FUNCTION_BLOCK L3_ProcessPlan (* Composite Function Block Type *)
  (* Standard: 61499-2 *)
  (* Version 0.0, 2014-10-13, EQUEROL, UJI *)
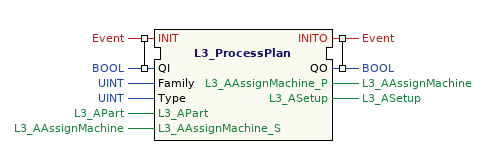
  EVENT_INPUT
    INIT WITH QI; (* Initialization Request *)
  END_EVENT
  EVENT_OUTPUT
    INITO WITH QO; (* Initialization Confirm *)
  END_EVENT
  VAR_INPUT
    QI : BOOL; (* Input event qualifier *)
    Family : UINT; (* Process plan family *)
    Type : UINT; (* Process plan type *)
  END_VAR
  VAR_OUTPUT
    QO : BOOL; (* Output event qualifier *)
  END_VAR
  SOCKETS
    L3_APart : L3_APart;
    L3_AAssignMachine_S : L3_AAssignMachine;
  END_SOCKETS
  PLUGS
    L3_AAssignMachine_P : L3_AAssignMachine;
    L3_ASetup : L3_ASetup;
  END_PLUGS
  FBS
    L3_PPTable : L3_PPTable;
    L3_NewPartHDLR : L3_NewPartHDLR;
    L3_MachineAllocator : L3_MachineAllocator;
    L3_MachineChecker : L3_MachineChecker;
    L3_CompletedPartHDLR : L3_CompletedPartHDLR;
    E_DELAY : E_DELAY;
    L3_SetupTable : L3_SetupTable;
    E_DELAY_1 : E_DELAY;
    L3_CompletedSetupHDLR_1 : L3_CompletedSetupHDLR;
  END_FBS
  EVENT_CONNECTIONS
    L3_AAssignMachine_S.CHK TO L3_MachineChecker.REQ;
    L3_MachineChecker.IND TO L3_PPTable.REQ;
    L3_PPTable.CNF TO L3_MachineChecker.RSP;
    L3_MachineChecker.CNF TO L3_AAssignMachine_P.CHK;
    L3_AAssignMachine_S.ASG TO L3_MachineAllocator.REQ;
    L3_MachineAllocator.Start TO E_DELAY.START;
    L3_MachineAllocator.Stop TO E_DELAY.STOP;
    E_DELAY.EO TO L3_MachineAllocator.Timeout;
    L3_MachineAllocator.CNF TO L3_AAssignMachine_P.ASG;
    L3_MachineAllocator.IND1 TO L3_SetupTable.REQ;
    L3_ASetup.CNF TO L3_MachineAllocator.RSP1;
    L3_MachineAllocator.IND2 TO L3_PPTable.REQ2;
    L3_PPTable.CNF2 TO L3_MachineAllocator.RSP2;
    L3_PPTable.CNF TO L3_MachineAllocator.REQ2;
    L3_SetupTable.CNF TO L3_ASetup.REQ;
    L3_APart.REQ TO L3_NewPartHDLR.REQ1;
    L3_NewPartHDLR.CNF1 TO L3_APart.CNF;
    L3_PPTable.IND1 TO L3_NewPartHDLR.REQ2;
    L3_NewPartHDLR.CNF2 TO L3_PPTable.RSP1;
    L3_CompletedPartHDLR.Start TO E_DELAY_1.START;
    L3_CompletedPartHDLR.Stop TO E_DELAY_1.STOP;
    E_DELAY_1.EO TO L3_CompletedPartHDLR.Timeout;
    L3_CompletedPartHDLR.CNF TO L3_PPTable.RSP3;
    L3_PPTable.IND3 TO L3_CompletedPartHDLR.REQ;
    L3_CompletedPartHDLR.IND TO L3_APart.IND;
    L3_APart.RSP TO L3_CompletedPartHDLR.RSP;
    L3_CompletedPartHDLR.INITO TO L3_PPTable.INIT;
    INIT TO L3_CompletedPartHDLR.INIT;
    L3_PPTable.INITO TO L3_SetupTable.INIT;
    L3_SetupTable.INITO TO INITO;
    L3_CompletedSetupHDLR_1.CNF1 TO L3_PPTable.RSP2;
    L3_PPTable.IND2 TO L3_CompletedSetupHDLR_1.REQ1;
    L3_ASetup.IND TO L3_CompletedSetupHDLR_1.REQ;
    L3_CompletedSetupHDLR_1.CNF TO L3_ASetup.RSP;
  END_CONNECTIONS
  DATA_CONNECTIONS
    L3_AAssignMachine_S.MTypeP TO L3_MachineChecker.MTypeIn;
    L3_AAssignMachine_S.MStateP TO L3_MachineChecker.MStateIn;
    L3_AAssignMachine_S.MPriorityP TO L3_MachineChecker.MPriorityIn;
    L3_AAssignMachine_S.MAssignP TO L3_MachineChecker.MAssignIn;
    L3_MachineChecker.MTypeOut TO L3_AAssignMachine_P.MTypeP;
    L3_MachineChecker.MStateOut TO L3_AAssignMachine_P.MStateP;
    L3_MachineChecker.MPriorityOut TO L3_AAssignMachine_P.MPriorityP;
    L3_MachineChecker.MAssignOut TO L3_AAssignMachine_P.MAssignP;
    L3_PPTable.vPriority TO L3_MachineChecker.Priority;
    L3_MachineAllocator.Delay TO E_DELAY.DT;
    L3_AAssignMachine_S.MFinalAssignP TO L3_MachineAllocator.MFinalAssignIn;
    L3_MachineAllocator.MFinalAssignOut TO L3_AAssignMachine_P.MFinalAssignP;
    L3_PPTable.vPartIDOut TO L3_MachineChecker.PartID;
    L3_PPTable.vPartIDOut TO L3_MachineAllocator.PartIDIn;
    L3_PPTable.vSetup TO L3_MachineAllocator.SetupIDIn;
    L3_MachineAllocator.PartIDOut TO L3_SetupTable.PartID;
    L3_MachineAllocator.SetupID TO L3_SetupTable.SetupID;
    L3_MachineAllocator.MID TO L3_SetupTable.MID;
    L3_SetupTable.PartInfo TO L3_ASetup.PartInfoP;
    L3_SetupTable.MID2 TO L3_ASetup.MID;
    L3_SetupTable.OPIDS TO L3_ASetup.OPIDS;
    L3_SetupTable.OPParams TO L3_ASetup.OPParams;
    L3_SetupTable.Fixture TO L3_ASetup.Fixture;
    L3_MachineAllocator.PartIDOut TO L3_PPTable.PartIDIn3;
    L3_MachineAllocator.MID TO L3_PPTable.MID;
    L3_APart.PartIDP TO L3_NewPartHDLR.PartIDIn;
    L3_APart.Lotsize TO L3_NewPartHDLR.LotsizeIn;
    L3_APart.Deadline TO L3_NewPartHDLR.DeadlineIn;
    L3_NewPartHDLR.PartIDOut TO L3_PPTable.PartIDIn1;
    L3_NewPartHDLR.LotsizeOut TO L3_PPTable.LotsizeIn;
    L3_NewPartHDLR.DeadlineOut TO L3_PPTable.DeadlineIn1;
    L3_CompletedPartHDLR.Delay TO E_DELAY_1.DT;
    L3_APart.Deadline TO L3_CompletedPartHDLR.DeadlineIn;
    L3_PPTable.PartIDOut TO L3_CompletedPartHDLR.PartIDIn;
    L3_AAssignMachine_S.MTypeP TO L3_PPTable.MType;
    L3_CompletedPartHDLR.QO TO L3_PPTable.QI;
    L3_CompletedPartHDLR.PartIDOut TO L3_APart.PartIDS;
    L3_CompletedPartHDLR.FamilyOut TO L3_APart.FamilyS;
    L3_CompletedPartHDLR.TypeOut TO L3_APart.TypeS;
    L3_CompletedPartHDLR.DeadlineOut TO L3_PPTable.DeadlineIn2;
    QI TO L3_CompletedPartHDLR.QI;
    Family TO L3_CompletedPartHDLR.FamilyIn;
    Type TO L3_CompletedPartHDLR.TypeIn;
    L3_PPTable.QO TO L3_SetupTable.QI;
    Family TO L3_PPTable.Family;
    Type TO L3_PPTable.Type;
    Type TO L3_SetupTable.Type;
    Family TO L3_SetupTable.Family;
    L3_SetupTable.QO TO QO;
    L3_CompletedSetupHDLR_1.PartIDOut TO L3_PPTable.PartIDIn2;
    L3_ASetup.PartInfoS TO L3_CompletedSetupHDLR_1.PartInfo;
  END_CONNECTIONS
END_FUNCTION_BLOCK
